PROGRAM MAIN
VAR
	fbShutdown	:FB_ShutDown; // Safely shutdown feature
	fbUPS		:FB_SUPS_CX51x0; // UPS type for test use
END_VAR

fbUPS.shutdown_delay := T#3S;
fbShutdown(fbUPS := fbUPS);

END_PROGRAM

(* stored: Version 1.1.0.1, ProductVersion 3.1.4024.12
   POU MAIN: Id {3439cf08-9e7a-47a5-a9ff-46ff00f18327}, SpecialFunc None *)
